{attribute 'linkalways'} 
{attribute 'no_explicit_call' := 'This FB is a CLASS and must be accessed using methods or properties'}
{attribute 'enable_dynamic_creation'}
FUNCTION_BLOCK StructuredDatatypeAddedEvent EXTENDS Disposable IMPLEMENTS I_StructuredDatatypeAddedEvent
VAR
	_target : I_StructuredDatatype;
END_VAR

METHOD FB_init : BOOL
VAR_INPUT
	bInitRetains : BOOL; // if TRUE, the retain variables are initialized (warm start / cold start)
	bInCopyCode : BOOL;  // if TRUE, the instance afterwards gets moved into the copy code (online change)
	Target : I_StructuredDatatype;
END_VAR
This^._target := Target;
END_METHOD

PROPERTY PUBLIC Target : I_StructuredDatatype
GET
Target := _target;
END_GET
END_PROPERTY

END_FUNCTION_BLOCK

(* stored: Version 1.1.0.1, ProductVersion 3.1.4024.12
   POU StructuredDatatypeAddedEvent: Id {7207408a-69fa-01e8-2131-613248254526}, SpecialFunc None
   Folder Constructor: Id {8b9b51e3-6096-02af-152d-8e0f0ecb7109}
   Method FB_init: Id {8a51a45f-b2ca-0fff-3782-1bb2c7cf3d70}
   Property Target: Id {6dc25461-994f-000f-2f27-bd445e54d8df}
   Get Get: Id {ef906220-f25d-0bad-0c77-e9a4b68a7946} *)
